PROGRAM main
  VAR
    Stop AT %IX0.4 : BOOL;
    Start AT %IX0.3 : BOOL;
    B1 AT %IX0.0 : BOOL;
    B2 AT %IX0.1 : BOOL;
    B3 AT %IX0.2 : BOOL;
    H1 AT %QX0.0 : BOOL;
    H2 AT %QX0.1 : BOOL;
    H3 AT %QX0.2 : BOOL;
    H4 AT %QX0.3 : BOOL;
    H5 AT %QX0.4 : BOOL;
    SystemActive AT %QX0.5 : BOOL;
  END_VAR

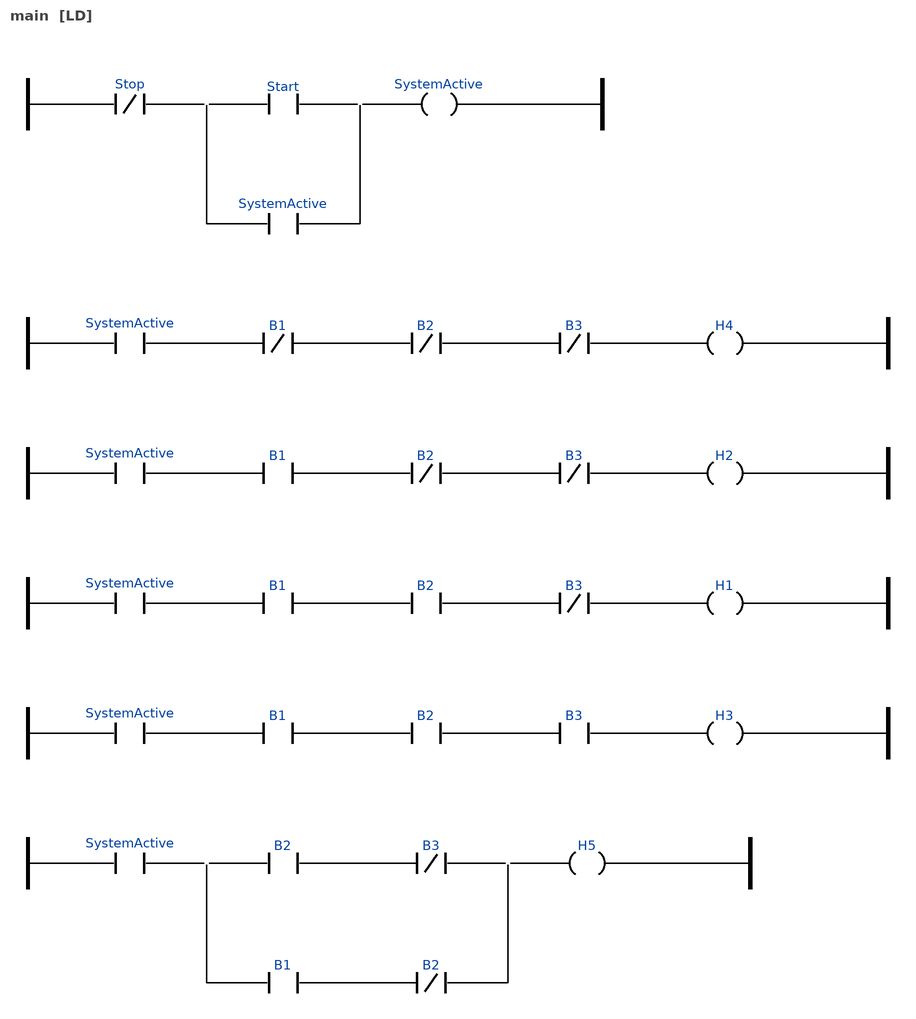
(* LD diagram, written out as Structured Text *)
SystemActive := NOT Stop AND (Start OR SystemActive);
H4 := SystemActive AND NOT B1 AND NOT B2 AND NOT B3;
H2 := SystemActive AND B1 AND NOT B2 AND NOT B3;
H1 := SystemActive AND B1 AND B2 AND NOT B3;
H3 := SystemActive AND B1 AND B2 AND B3;
H5 := SystemActive AND (B1 AND NOT B2 OR B2 AND NOT B3);
END_PROGRAM
